// TIA Portal V19 export
DATA_BLOCK "SET_PARAMETERS"   // DB24
{ S7_Optimized_Access := 'FALSE' }
   VAR RETAIN
      "RINSE-1_CLEANING_TIME_SV" : Int;
      "RINSE-1_CLEANING_TIME_PV" : Int;
      "RINSE-1_RECIRCULATION_TIME_SV" : Int;
      "RINSE-1_RECIRCULATION_TIME_PV" : Int;
      "RINSE-1_DRAIN_TIME_SV" : Int;
      "RINSE-1_DRAIN_TIME_PV" : Int;
      "RINSE-1_PUMP_CHASING_TIME_SV" : Int;
      "RINSE-1_PUMP_CHASING_TIME_PV" : Int;
      "RINSE-1_TEMPERATURE_SET" : Real;
      "RINSE-2_TEMPERATURE_SET" : Real;
      "RINSE-2_CLEANING_TIME_SV" : Int;
      "RINSE-2_CLEANING_TIME_PV" : Int;
      "RINSE-2_RECIRCULATION_TIME_SV" : Int;
      "RINSE-2_RECIRCULATION_TIME_PV" : Int;
      "RINSE-2_DRAIN_TIME_SV" : Int;
      "RINSE-2_DRAIN_TIME_PV" : Int;
      "RINSE-2_PUMP_CHASING_TIME_SV" : Int;
      "RINSE-2_PUMP_CHASING_TIME_PV" : Int;
      DOSING_TIME_SV : Int;
      DOSING_TIME_PV : Int;
      "ALKALI/ACID_TEMPERATURE_SET" : Real;
      "ALKALI/ACID_CLEANING_TIME_SV" : Int;
      "ALKALI/ACID_CLEANING_TIME_PV" : Int;
      "ALKALI/ACID_RECIRCULATION_TIME_SV" : Int;
      "ALKALI/ACID_RECIRCULATION_TIME_PV" : Int;
      "ALKALI/ACID_DRAIN_TIME_SV" : Int;
      "ALKALI/ACID_DRAIN_TIME_PV" : Int;
      "ALKALI/ACID_PUMP_CHASING_TIME_SV" : Int;
      "ALKALI/ACID_PUMP_CHASING_TIME_PV" : Int;
      FINAL_RINSE_TEMPERATURE_SET : Real;
      FINAL_RINSE_CLEANING_TIME_SV : Int;
      FINAL_RINSE_CLEANING_TIME_PV : Int;
      FINAL_RINSE_RECIRCULATION_TIME_SV : Int;
      FINAL_RINSE_RECIRCULATION_TIME_PV : Int;
      FINAL_RINSE_DRAIN_TIME_SV : Int;
      FINAL_RINSE_DRAIN_TIME_PV : Int;
      FINAL_RINSE_PUMP_CHASING_TIME_SV : Int;
      FINAL_RINSE_PUMP_CHASING_TIME_PV : Int;
      CONDUCTIVITY_SET : Real;
      PH_SET : Real;
      DOSING_PH_LOW : Real;
      DOSING_PH_HIGH : Real;
      "RINSE-3_TEMPERATURE_SET" : Real;
      "RINSE-3_CLEANING_TIME_SV" : Int;
      "RINSE-3_CLEANING_TIME_PV" : Int;
      "RINSE-3_RECIRCULATION_TIME_SV" : Int;
      "RINSE-3_RECIRCULATION_TIME_PV" : Int;
      "RINSE-3_DRAIN_TIME_SV" : Int;
      "RINSE-3_DRAIN_TIME_PV" : Int;
      "RINSE-3_PUMP_CHASING_TIME_SV" : Int;
      "RINSE-3_PUMP_CHASING_TIME_PV" : Int;
      SET_TEMPERATURE : Real;
      "RINSE-1_FWD_PUMP_HEATING_RPM" : Int;
      "RINSE-1_FWD_PUMP_CLEANING_RPM" : Int;
      "RINSE-2_FWD_PUMP_HEATING_RPM" : Int;
      "RINSE-2_FWD_PUMP_CLEANING_RPM" : Int;
      "ALKALI/ACID_FWD_PUMP_HEATING_RPM" : Int;
      "ALKALI/ACID_FWD_PUMP_CLEANING_RPM" : Int;
      "FINAL_RINSE-2_FWD_PUMP_HEATING_RPM" : Int;
      "FINAL_RINSE-2_FWD_PUMP_CLEANING_RPM" : Int;
      "FINAL_RINSE-1_FWD_PUMP_HEATING_RPM" : Int;
      "FINAL_RINSE-1_FWD_PUMP_CLEANING_RPM" : Int;
      "PUMP-1_SPEED" : Int;
      RECIRCULATION_PH_LOW : Real;
      RECIRCULATION_PH_HIGH : Real;
      PLANT1_TANK_SELECT : Byte;
      PLANT_SELECT : Byte;
      PLANT2_TANK_SELECT : Byte;
      PLANT3_TANK_SELECT : Byte;
      "SW TANK_CLEANING_TIME_SV" : Int;
      "SW TANK_CLEANING_TIME_PV" : Int;
      "SW TANK_DRAIN_TIME_SV" : Int;
      "SW TANK_DRAIN_TIME_PV" : Int;
      "SW TANK_PUMP_CHASING_TIME_SV" : Int;
      "SW TANK_PUMP_CHASING_TIME_PV" : Int;
      "PW TANK_CLEANING_TIME_SV" : Int;
      "PW TANK_CLEANING_TIME_PV" : Int;
      "PW TANK_DRAIN_TIME_SV" : Int;
      "PW TANK_DRAIN_TIME_PV" : Int;
      "PW TANK_PUMP_CHASING_TIME_SV" : Int;
      "PW TANK_PUMP_CHASING_TIME_PV" : Int;
      "SW TANK_FWD_PUMP_CLEANING_RPM" : Int;
      "PW TANK_FWD_PUMP_CLEANING_RPM" : Int;
      "SW TANK_TEMPERATURE_SET" : Real;
      "PW TANK_TEMPERATURE_SET" : Real;
      DOSING_PH_LOW1 : Real;
      DOSING_PH_HIGH1 : Real;
   END_VAR
BEGIN
END_DATA_BLOCK
